(* CoDeSys 2.3 export: GARDEROBA.EXP *)

(* POU Rooms/Garderoba, ST *)
FUNCTION_BLOCK Garderoba
VAR
	mainLampG:OnOff;
END_VAR
mainLampG(input:=H3_1b, output => G3_1);
END_FUNCTION_BLOCK
